// TIA Portal project "Project1" (V18)

(* hardware
DEVICE "S7-1200 station_1"  S7-1200 Station
   slot 0: "Rack_0"  S7-1200 Rack  Rack  V1.0
   slot 1: "PLC_1"  CPU 1215C AC/DC/Rly  6ES7 215-1BG40-0XB0  V4.6
*)

// ===== PLC "PLC_1"  CPU 1215C AC/DC/Rly =====

VAR_GLOBAL   // PLC tag table "Default tag table"
   "START" AT %I0.0 : Bool;
   "STOP" AT %I0.1 : Bool;
   "EMERGENCY STOP" AT %I0.2 : Bool;
   "MOTOR1" AT %Q0.3 : Bool;
   "MOTOR2" AT %Q0.4 : Bool;
   "MOTOR3" AT %Q0.5 : Bool;
   "LAMB1" AT %Q0.6 : Bool;
   "LAMB2" AT %Q0.7 : Bool;
   "LAMB3" AT %Q1.0 : Bool;
   "ALARM" AT %Q1.1 : Bool;
   "Tag_1" AT %M5.0 : Bool;
END_VAR

// folder: System blocks/Program resources

DATA_BLOCK "Data_block_1"   // DB1
{ S7_Optimized_Access := 'TRUE' }
AUTHOR : Simatic
FAMILY : IEC
NAME : IEC_TMR
VERSION : 1.0
// stored: InstanceOfName IEC_TIMER
"IEC_TIMER"
BEGIN
END_DATA_BLOCK

// folder: (top level)

ORGANIZATION_BLOCK "Main"   // OB1, LAD, ProgramCycle
TITLE = "Main Program Sweep (Cycle)"
{ S7_Optimized_Access := 'TRUE' }
VERSION : 0.1
   VAR_INPUT
      Initial_Call : Bool;   // Initial call of this OB
      Remanence : Bool;   // =True, if remanent data are available
   END_VAR
BEGIN

REGION Network 1
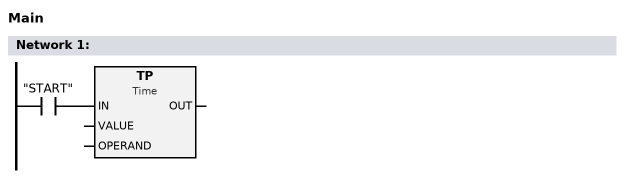
   // no checked SCL form for this network; see the picture
END_REGION
END_ORGANIZATION_BLOCK